FUNCTION_BLOCK Sequence1Task EXTENDS TcoCore.TcoTask
VAR_INPUT
	Sequence : TcoCore.ITcoSequencer;
END_VAR

(*~
	<docu>
		<summary>
			Restores this instance to the Ready state. Can be called explicitly or from within one of the restore mechanisms.
			<para>
				See also <see cref="PlcDocu.TcoCore.TcoTask.AutoRestorable()"/>
			</para>
		</summary>			
	</docu>	
~*)
METHOD Restore : ITcoRestorable
SUPER^.Restore();
THIS^.Sequence.Restore();
END_METHOD

END_FUNCTION_BLOCK

(* stored: Version 1.1.0.1, ProductVersion 3.1.4024.12
   POU Sequence1Task: Id {9ca577a3-fab9-0e8f-3ad3-b338c0857701}, SpecialFunc None
   Method Restore: Id {a30a6bcb-6e73-0d33-1d97-c339684551b5} *)
